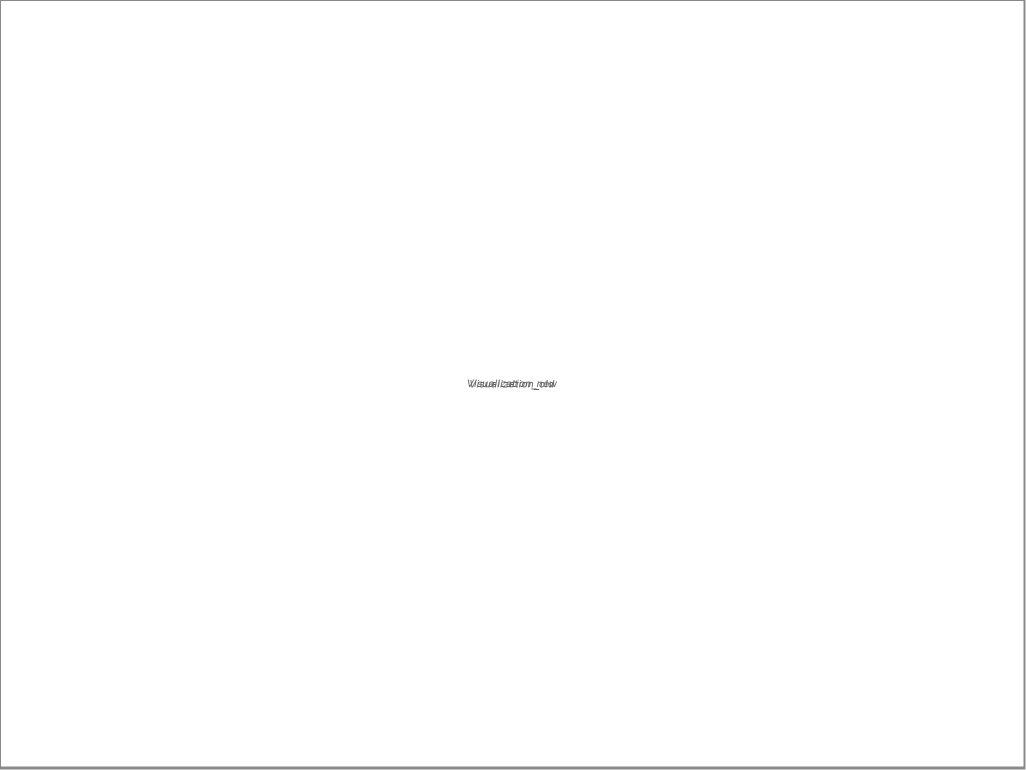
VISUALIZATION Visualization  // 1026x770
    Frame (0,0 1024x768), invisible if: GVL.bRegiFelulet=FALSE, input disabled if: GVL.bRegiFelulet=FALSE
        shows Visualization_old()
    Frame (0,0 1024x767), invisible if: GVL.bRegiFelulet, input disabled if: GVL.bRegiFelulet
        shows Visualization_new()
END_VISUALIZATION

(* stored: Version 1.1.0.1, ProductVersion 3.1.4024.11
   Visu Visualization: Id {ef1c286a-e38e-4e00-85bd-d246715f9b7d} *)
